FUNCTION_BLOCK FB_NOTT_BIREFRINGENCE
VAR_INPUT
END_VAR
VAR_OUTPUT
END_VAR
VAR
	NPC1:		FB_NOTT_MOTOR;
	NPC2:		FB_NOTT_MOTOR;
	NPC3:		FB_NOTT_MOTOR;
	NPC4:		FB_NOTT_MOTOR;
	
	
	ptrNPCs:	ARRAY [1..4] OF POINTER TO FB_NOTT_MOTOR;
	// GUI stuff
	guiNPCsIndex:	UINT := 1;	// Index for Shutter Engineering GUI
	
	stat:		T_NOTT_STAT;
	
END_VAR



NPC1(
	in_bSafe:=, 
	in_bDisableIfUnsafe:=, 
	sName:= 'NPC 1', 
	nNOVRAM_DevId:= 6, 
	nNOVRAM_Offset:= 33000);
	
NPC2(
	in_bSafe:=, 
	in_bDisableIfUnsafe:=, 
	sName:= 'NPC 2', 
	nNOVRAM_DevId:= 6, 
	nNOVRAM_Offset:= 34000);
	
NPC3(
	in_bSafe:=, 
	in_bDisableIfUnsafe:=, 
	sName:= 'NPC 3', 
	nNOVRAM_DevId:= 6, 
	nNOVRAM_Offset:= 35000);
	
NPC4(
	in_bSafe:=, 
	in_bDisableIfUnsafe:=, 
	sName:= 'NPC 4', 
	nNOVRAM_DevId:= 6, 
	nNOVRAM_Offset:= 36000);

	
M_Configure();

METHOD M_Configure : BOOL
VAR_INPUT
END_VAR

ptrNPCs[1] := ADR(NPC1);
ptrNPCs[2] := ADR(NPC2);
ptrNPCs[3] := ADR(NPC3);
ptrNPCs[4] := ADR(NPC4);
END_METHOD

END_FUNCTION_BLOCK

(* stored: Version 1.1.0.1, ProductVersion 3.1.4024.14
   POU FB_NOTT_BIREFRINGENCE: Id {d8ffa56c-39eb-4490-bea3-43e42a3155cd}, SpecialFunc None
   Method M_Configure: Id {b159d3b8-ea9a-4672-9768-4b0e2d61c266} *)
